// TIA Portal project "LAP_2010_4_Abfuellanlage" (V14)

(* hardware
DEVICE "S7-1200-Station_1"  S7-1200 Station
   slot 0: "Baugruppenträger_0"  S7-1200 Rack  Rack  V1.0
   slot 1: "PLC_1"  CPU 1214C DC/DC/DC  6ES7 214-1AG40-0XB0  V4.2
   slot 3: "AQ 1x12BIT_1"  AQ1 signal board  6ES7 232-4HA30-0XB0  V1.0
*)

// ===== PLC "PLC_1"  CPU 1214C DC/DC/DC =====

VAR_GLOBAL   // PLC tag table "Standard-Variablentabelle"
   "System_Byte" AT %MB100 : Byte;
   "FirstScan" AT %M100.0 : Bool;
   "DiagStatusUpdate" AT %M100.1 : Bool;
   "AlwaysTRUE" AT %M100.2 : Bool;
   "AlwaysFALSE" AT %M100.3 : Bool;
   "Clock_Byte" AT %MB110 : Byte;
   "Clock_10Hz" AT %M110.0 : Bool;
   "Clock_5Hz" AT %M110.1 : Bool;
   "Clock_2.5Hz" AT %M110.2 : Bool;
   "Clock_2Hz" AT %M110.3 : Bool;
   "Clock_1.25Hz" AT %M110.4 : Bool;
   "Clock_1Hz" AT %M110.5 : Bool;
   "Clock_0.625Hz" AT %M110.6 : Bool;
   "Clock_0.5Hz" AT %M110.7 : Bool;
   "Q1" AT %Q0.0 : Bool;
   "Q2" AT %Q0.1 : Bool;
   "S1" AT %I0.0 : Bool;
   "S2" AT %I0.1 : Bool;
   "S3" AT %I0.2 : Bool;
   "S4" AT %I0.3 : Bool;
   "S5" AT %I0.4 : Bool;
   "AlleAusgänge" AT %QW0 : Word;
   "Q3" AT %Q0.2 : Bool;
   "Q4" AT %Q0.3 : Bool;
   "Q5" AT %Q0.4 : Bool;
   "Q6" AT %Q0.5 : Bool;
END_VAR

DATA_BLOCK "DigInput"   // DB1
{ S7_Optimized_Access := 'FALSE' }
VERSION : 0.1
   VAR
      S1 : Bool;   // Taster "Reset"
      S2 : Bool;   // Taster "Start"
      S7 : Bool;   // Füllstand
      S8 : Bool;   // Position Dose
   END_VAR
BEGIN
END_DATA_BLOCK

DATA_BLOCK "DigOutput"   // DB2
{ S7_Optimized_Access := 'FALSE' }
VERSION : 0.1
   VAR
      K1 : Bool;   // Antrieb Förderband
      K2 : Bool;   // Spule Vereinzelner
      K3 : Bool;   // Spule Füllen
      H2 : Bool;   // Meldeleuchte "Behälter leer"
   END_VAR
BEGIN
END_DATA_BLOCK

ORGANIZATION_BLOCK "Main"   // OB1, LAD, ProgramCycle
TITLE = "Main Program Sweep (Cycle)"
{ S7_Optimized_Access := 'TRUE' }
VERSION : 0.1
   VAR_INPUT
      Initial_Call : Bool;   // Initial call of this OB
      Remanence : Bool;   // =True, if remanent data are available
   END_VAR
BEGIN

REGION Network 1: Ventil Tank 1 unten
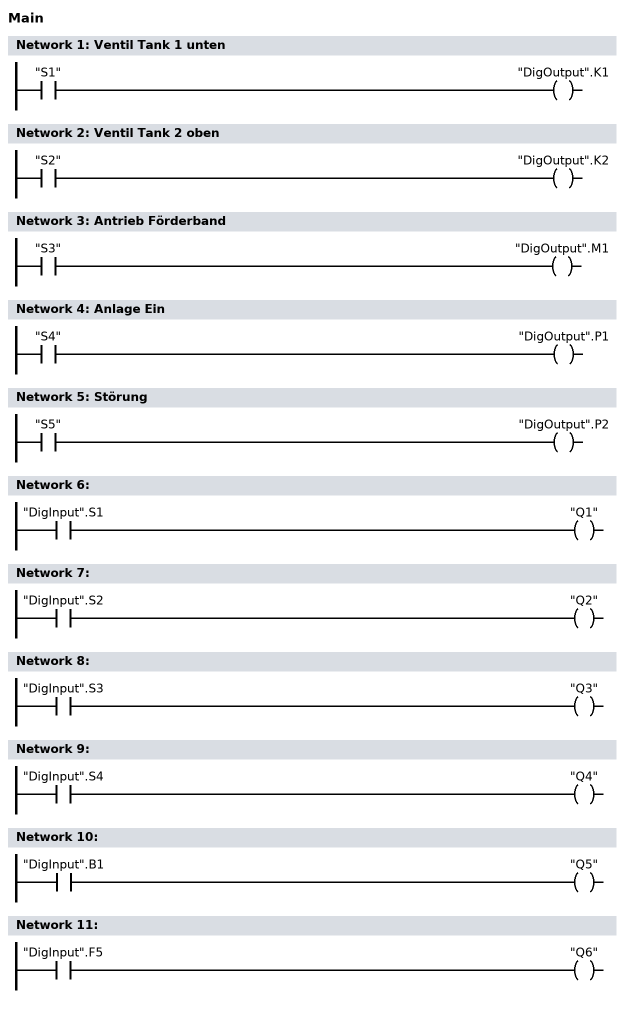
   RUNG wire#powerrail
      Contact( "S1" )
      Coil( "DigOutput".K1 )
   END_RUNG
   // the same network as SCL:
   "DigOutput".K1 := "S1";
END_REGION

REGION Network 2: Ventil Tank 2 oben
   RUNG wire#powerrail
      Contact( "S2" )
      Coil( "DigOutput".K2 )
   END_RUNG
   // the same network as SCL:
   "DigOutput".K2 := "S2";
END_REGION

REGION Network 3: Antrieb Förderband
   RUNG wire#powerrail
      Contact( "S3" )
      Coil( "DigOutput".M1 )
   END_RUNG
   // the same network as SCL:
   "DigOutput".M1 := "S3";
END_REGION

REGION Network 4: Anlage Ein
   RUNG wire#powerrail
      Contact( "S4" )
      Coil( "DigOutput".P1 )
   END_RUNG
   // the same network as SCL:
   "DigOutput".P1 := "S4";
END_REGION

REGION Network 5: Störung
   RUNG wire#powerrail
      Contact( "S5" )
      Coil( "DigOutput".P2 )
   END_RUNG
   // the same network as SCL:
   "DigOutput".P2 := "S5";
END_REGION

REGION Network 6
   RUNG wire#powerrail
      Contact( "DigInput".S1 )
      Coil( "Q1" )
   END_RUNG
   // the same network as SCL:
   "Q1" := "DigInput".S1;
END_REGION

REGION Network 7
   RUNG wire#powerrail
      Contact( "DigInput".S2 )
      Coil( "Q2" )
   END_RUNG
   // the same network as SCL:
   "Q2" := "DigInput".S2;
END_REGION

REGION Network 8
   RUNG wire#powerrail
      Contact( "DigInput".S3 )
      Coil( "Q3" )
   END_RUNG
   // the same network as SCL:
   "Q3" := "DigInput".S3;
END_REGION

REGION Network 9
   RUNG wire#powerrail
      Contact( "DigInput".S4 )
      Coil( "Q4" )
   END_RUNG
   // the same network as SCL:
   "Q4" := "DigInput".S4;
END_REGION

REGION Network 10
   RUNG wire#powerrail
      Contact( "DigInput".B1 )
      Coil( "Q5" )
   END_RUNG
   // the same network as SCL:
   "Q5" := "DigInput".B1;
END_REGION

REGION Network 11
   RUNG wire#powerrail
      Contact( "DigInput".F5 )
      Coil( "Q6" )
   END_RUNG
   // the same network as SCL:
   "Q6" := "DigInput".F5;
END_REGION
END_ORGANIZATION_BLOCK

ORGANIZATION_BLOCK "Startup"   // OB100, SCL, Startup
TITLE = "Complete Restart"
{ S7_Optimized_Access := 'TRUE' }
VERSION : 0.1
   VAR_INPUT
      LostRetentive : Bool;   // True if retentive data are lost
      LostRTC : Bool;   // True if date and time are lost
   END_VAR
BEGIN
   "AlleAusgänge" := 16#0000;
END_ORGANIZATION_BLOCK